% RSLogix 500 project WATER TANK FILLING CONTROL LOGIC_BAK005.RSS, saved by version 8.30.00.16 %
PROJECT "UNTITLED"    % processor: Bul.1763 MicroLogix 1100 Series B %

PROGRAM FILES
  LAD 2   4 rungs

DATA FILES
  O0 OUTPUT  4 elements
  I1 INPUT  6 elements
  S2 STATUS  66 elements
  B3 BINARY  1 elements
  T4 TIMER  1 elements
  C5 COUNTER  1 elements
  R6 CONTROL  1 elements
  N7 INTEGER  1 elements
  F8 FLOAT  1 elements

LADDER 2
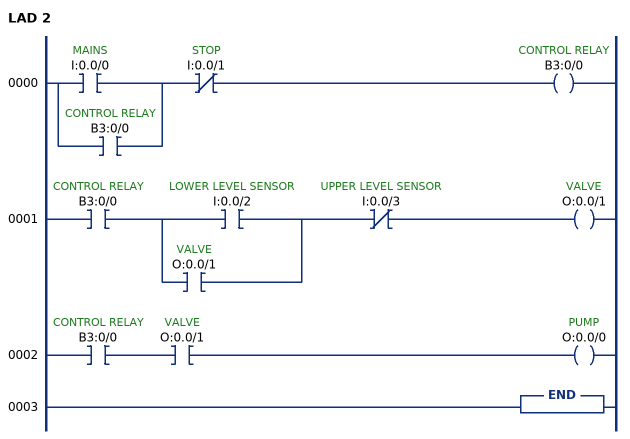
% Rung: 0 %
SOR BST XIC I:0.0/0 NXB XIC B3:0/0 BND XIO I:0.0/1 OTE B3:0/0 EOR
%   I:0.0/0  "MAINS" %
%   B3:0/0  "CONTROL RELAY" %
%   I:0.0/1  "STOP" %
% Rung: 1 %
SOR XIC B3:0/0 BST XIC I:0.0/2 NXB XIC O:0.0/1 BND XIO I:0.0/3 OTE O:0.0/1 EOR
%   B3:0/0  "CONTROL RELAY" %
%   I:0.0/2  "LOWER LEVEL SENSOR" %
%   O:0.0/1  "VALVE" %
%   I:0.0/3  "UPPER LEVEL SENSOR" %
% Rung: 2 %
SOR XIC B3:0/0 XIC O:0.0/1 OTE O:0.0/0 EOR
%   B3:0/0  "CONTROL RELAY" %
%   O:0.0/1  "VALVE" %
%   O:0.0/0  "PUMP" %
% Rung: 3 %
SOR END EOR

DATA TABLE (non-zero values as saved)
DATA B3
% B3:0 % 0X0001
